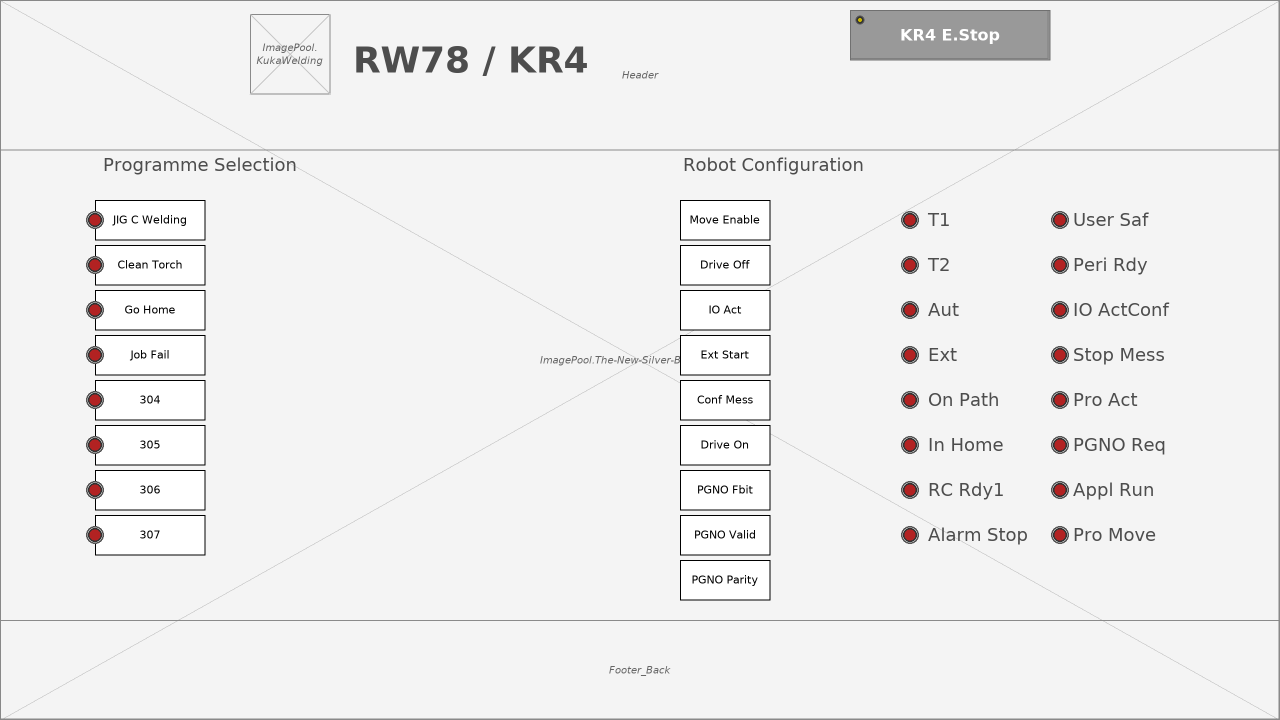
VISUALIZATION PAGE_KR4  // 1280x720
    Image (0,0 1280x720), image: ImagePool.The-New-Silver-Backgrounds
    Frame (0,620 1280x100)
        shows Footer_Back()
    Frame (0,0 1280x150)
        shows Header()
    Image (250,14 80x80), image: ImagePool.KukaWelding
    Label (350,40 300x40), "RW78 / KR4"
    Label (100,150 200x30), "Programme Selection"
    RoundedRectangle (680,200 90x40), "Move Enable"
        toggle KR4.bOutBit[1,0]
    RoundedRectangle (680,245 90x40), "Drive Off"
        toggle KR4.bOutBit[1,1]
    RoundedRectangle (680,290 90x40), "IO Act"
        toggle KR4.bOutBit[1,2]
    RoundedRectangle (680,335 90x40), "Ext Start"
        toggle KR4.bOutBit[1,3]
    RoundedRectangle (680,380 90x40), "Conf Mess"
        toggle KR4.bOutBit[1,4]
    RoundedRectangle (680,425 90x40), "Drive On"
        toggle KR4.bOutBit[1,5]
    RoundedRectangle (680,470 90x40), "PGNO Fbit"
        toggle KR4.bOutBit[1,6]
    RoundedRectangle (680,515 90x40), "PGNO Valid"
        toggle KR4.bOutBit[1,7]
    RoundedRectangle (680,560 90x40), "PGNO Parity"
        toggle KR4.bOutBit[2,0]
    Label (680,150 200x30), "Robot Configuration"
    Lamp1 (900,210 20x20), variable: KR4.bInBit[1,0], style: Lamp-Lamp1-Red
    Lamp1 (900,255 20x20), variable: KR4.bInBit[1,1], style: Lamp-Lamp1-Red
    Lamp1 (900,300 20x20), variable: KR4.bInBit[1,2], style: Lamp-Lamp1-Red
    Lamp1 (900,345 20x20), variable: KR4.bInBit[1,3], style: Lamp-Lamp1-Red
    Lamp1 (900,390 20x20), variable: KR4.bInBit[1,4], style: Lamp-Lamp1-Red
    Lamp1 (900,435 20x20), variable: KR4.bInBit[1,5], style: Lamp-Lamp1-Red
    Lamp1 (900,480 20x20), variable: KR4.bInBit[1,6], style: Lamp-Lamp1-Red
    Lamp1 (900,525 20x20), variable: KR4.bInBit[1,7], style: Lamp-Lamp1-Red
    Lamp1 (1050,210 20x20), variable: KR4.bInBit[2,0], style: Lamp-Lamp1-Red
    Lamp1 (1050,255 20x20), variable: KR4.bInBit[2,1], style: Lamp-Lamp1-Red
    Lamp1 (1050,300 20x20), variable: KR4.bInBit[2,2], style: Lamp-Lamp1-Red
    Lamp1 (1050,345 20x20), variable: KR4.bInBit[2,3], style: Lamp-Lamp1-Red
    Lamp1 (1050,390 20x20), variable: KR4.bInBit[2,4], style: Lamp-Lamp1-Red
    Lamp1 (1050,435 20x20), variable: KR4.bInBit[2,5], style: Lamp-Lamp1-Red
    Lamp1 (1050,480 20x20), variable: KR4.bInBit[2,6], style: Lamp-Lamp1-Red
    Lamp1 (1050,525 20x20), variable: KR4.bInBit[2,7], style: Lamp-Lamp1-Red
    Group (850,10 200x50)
        Button (0,0 200x50), "KR4 E.Stop"
            toggle KR4.KR4_Estop
        Lamp1 (5,5 10x10), variable: KR4.KR4_Estop, style: Lamp-Lamp1-Yellow
    Label (1070,205 110x30), "User Saf"
    Label (1070,250 110x30), "Peri Rdy"
    Label (1070,295 110x30), "IO ActConf"
    Label (1070,340 110x30), "Stop Mess"
    Label (1070,385 110x30), "Pro Act"
    Label (1070,430 110x30), "PGNO Req"
    Label (1070,475 110x30), "Appl Run"
    Label (1070,520 110x30), "Pro Move"
    Label (925,205 105x30), "T1"
    Label (925,250 105x30), "T2"
    Label (925,295 105x30), "Aut"
    Label (925,340 105x30), "Ext"
    Label (925,385 105x30), "On Path"
    Label (925,430 105x30), "In Home"
    Label (925,475 105x30), "RC Rdy1"
    Label (925,520 105x30), "Alarm Stop"
    RoundedRectangle (95,200 110x40), "JIG C Welding"
        toggle KR4.bOutBit[3,0]
    RoundedRectangle (95,245 110x40), "Clean Torch"
        toggle KR4.bOutBit[3,1]
    RoundedRectangle (95,290 110x40), "Go Home"
        toggle KR4.bOutBit[3,2]
    RoundedRectangle (95,335 110x40), "Job Fail"
        toggle KR4.bOutBit[3,3]
    RoundedRectangle (95,380 110x40), "304"
        toggle KR4.bOutBit[3,4]
    RoundedRectangle (95,425 110x40), "305"
        toggle KR4.bOutBit[3,5]
    RoundedRectangle (95,470 110x40), "306"
        toggle KR4.bOutBit[3,6]
    RoundedRectangle (95,515 110x40), "307"
        toggle KR4.bOutBit[3,7]
    Lamp1 (85,210 20x20), variable: KR4.bInBit[3,0], style: Lamp-Lamp1-Red
    Lamp1 (85,255 20x20), variable: KR4.bInBit[3,1], style: Lamp-Lamp1-Red
    Lamp1 (85,300 20x20), variable: KR4.bInBit[3,2], style: Lamp-Lamp1-Red
    Lamp1 (85,345 20x20), variable: KR4.bInBit[3,3], style: Lamp-Lamp1-Red
    Lamp1 (85,390 20x20), variable: KR4.bInBit[3,4], style: Lamp-Lamp1-Red
    Lamp1 (85,435 20x20), variable: KR4.bInBit[3,5], style: Lamp-Lamp1-Red
    Lamp1 (85,480 20x20), variable: KR4.bInBit[3,6], style: Lamp-Lamp1-Red
    Lamp1 (85,525 20x20), variable: KR4.bInBit[3,7], style: Lamp-Lamp1-Red
END_VISUALIZATION

(* stored: Version 1.1.0.1, ProductVersion 3.1.4024.12
   Visu PAGE_KR4: Id {539150db-6a44-4998-9251-2f927c3fa0da} *)
